# EPICS substitutions: iocBoot/ioc-xpp-gige-01/ioc-xpp-gige-01.substitutions
#
# GigE IOC archive substitutions file
#

# Generate IOC archive request
file archive_gige.archive
{
    {
        IOC = IOC:XPP:GIGE:01,
    }
}
